INTERFACE I_State

METHOD SafetyAcknowledged
VAR_INPUT
END_VAR
END_METHOD

METHOD SafetyTripped
VAR_INPUT
END_VAR
END_METHOD

METHOD StartButtonPressed
END_METHOD

METHOD StopButtonPressed
END_METHOD

END_INTERFACE

(* stored: Version 1.1.0.1, ProductVersion 3.1.4024.11
   Itf I_State: Id {9cabd902-5128-4a1b-870f-67fd091ef023}
   Method SafetyAcknowledged: Id {521727b2-f658-4259-9626-8155edba540d}
   Method SafetyTripped: Id {e9e19173-0a98-4f7d-9f1a-b489646f2a63}
   Method StartButtonPressed: Id {c27a95ed-7eb3-4ce2-a499-f52fe471f04c}
   Method StopButtonPressed: Id {5653cda2-2f42-4886-9fae-7114d7fb78d2} *)
